(* PLC project Unbenannt, Unbekannt Unbenannt 1 *)
(* stored: creationDateTime 2019-08-23T13:38:07, modificationDateTime 2019-09-16T21:40:09 *)

(* Output current execution time in miliseconds *)
FUNCTION T_PLC_MS : UDINT
  VAR
    tx : UDINT;
  END_VAR
  VAR_INPUT
    debug : BOOL;
  END_VAR
  VAR
    N : INT := 0;
    offset : UDINT := 0;
    temp : DWORD := 1;
  END_VAR

            tx := 0;

{extern unsigned long __tick;
extern unsigned long long common_ticktime__;
unsigned long long ticktime_ms = (common_ticktime__)/1000000;
UDINT plc_time = (UDINT)(ticktime_ms * (unsigned long long)__tick);
TX = plc_time}

T_PLC_MS := tx;
IF debug THEN
	T_PLC_MS := (DWORD_TO_UDINT(SHL(UDINT_TO_DWORD(T_PLC_MS),N) OR SHL(temp,N))-1) + OFFSET;
END_IF;

(* Original Code:
tx := TIME();
T_PLC_MS := TIME_TO_DWORD(Tx);
IF debug THEN
	T_PLC_MS := (SHL(T_PLC_MS,N) OR SHL(DWORD#1,N)-1) + OFFSET;
END_IF;
*)

(* From OSCAT library, www.oscat.de

this is a temporary T_PLC_MS FB until OpenPLC gets it´s own time() functionality *)

(* PLC_TIME and Global variables PLC_SCAN_CYCL and PLC_CYCL_TIME required *)
          
END_FUNCTION

FUNCTION_BLOCK F_POLY
  VAR_INPUT
    X : REAL;
    C : ARRAY[0..7] OF REAL;
  END_VAR
  VAR_OUTPUT
    _F_POLY : REAL;
  END_VAR

            _F_POLY := ((((((( c[7] * x + c[6] ) * x + c[5] ) * x + c[4] ) * x + c[3] ) * x + c[2] ) * x + c[1] ) * x + c[0] ) ;

          
END_FUNCTION_BLOCK

PROGRAM program0
  VAR
    LocalVar0 : DINT;
    LocalVar1 : DINT;
    LocalVar2 : DINT;
    LocalVar3 : REAL;
    F_POLY0 : F_POLY;
  END_VAR

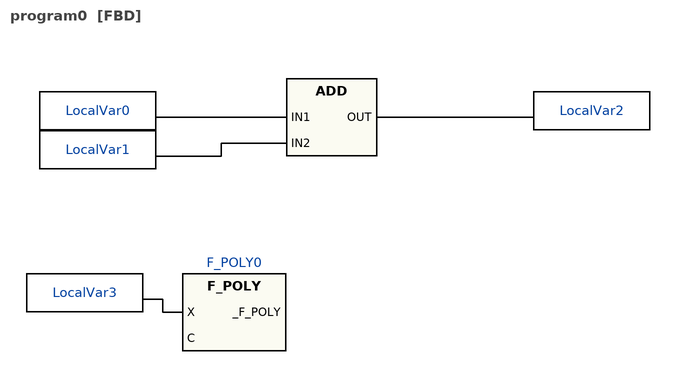
(* FBD diagram, written out as Structured Text *)
LocalVar2 := LocalVar0 + LocalVar1;
F_POLY0(X := LocalVar3);
END_PROGRAM

(* calculates the linear equation f_lin = a*x + b *)
FUNCTION F_LIN : REAL
  VAR_INPUT
    X : REAL;
    A : REAL;
    B : REAL;
  END_VAR

            F_lin := A * X + B;
(* from OSCAT library www.oscat.de *)
          
END_FUNCTION

(* this function calculates the linear equation f_lin = a*x + b given by two points x1/y1 and x2/y2 *)
FUNCTION F_LIN2 : REAL
  VAR_INPUT
    X : REAL;
    X1 : REAL;
    X2 : REAL;
    Y1 : REAL;
    Y2 : REAL;
  END_VAR

            F_LIN2 := (Y2 - Y1) / (X2 - X1) * (X - X1) + Y1;
(* from OSCAT library www.oscat.de *)
          
END_FUNCTION

(* calculates the power equation f_power = a*x^n *)
FUNCTION F_POWER : REAL
  VAR
    A : REAL;
    X : REAL;
    N : REAL;
  END_VAR

            f_power := a * EXPT(X,N);
(* from OSCAT library www.oscat.de *)
          
END_FUNCTION

(* calculates the quadratic equation f_lin = a*x + b *)
FUNCTION F_QUAD : REAL
  VAR
    X : REAL;
    A : REAL;
    B : REAL;
    C : REAL;
  END_VAR

            F_QUAD :=  (A * X + B) * X + C;
(* from OSCAT library www.oscat.de *)
          
END_FUNCTION

(* calculates a ramp and limits the output to 0 .. 255 without overflow problems *)
FUNCTION FRMP_B : BYTE
  VAR
    START : BYTE;
    DIR : BOOL;
    TD : TIME;
    TR : TIME;
  END_VAR

            IF TD < TR THEN
	FRMP_B := MIN(UDINT_TO_BYTE(DWORD_TO_UDINT(SHL(TIME_TO_DWORD(TD), 8)) / TIME_TO_UDINT(TR)), SEL(DIR, START, USINT_TO_BYTE(USINT#255 - BYTE_TO_USINT(START))));
	IF DIR THEN
		FRMP_B := USINT_TO_BYTE(BYTE_TO_USINT(START) + BYTE_TO_USINT(FRMP_B));
	ELSE
		FRMP_B := USINT_TO_BYTE(BYTE_TO_USINT(START) - BYTE_TO_USINT(FRMP_B));
	END_IF;
ELSE
	FRMP_B := SEL(DIR, BYTE#0, BYTE#255);
END_IF;
(* from OSCAT library www.oscat.de *)
          
END_FUNCTION

(* This is a increment function which increments the variable X by 1 and if N is reached, it begins with 0 instead of N again. *)
FUNCTION INC1 : INT
  VAR_INPUT
    X : INT;
    N : INT;
  END_VAR

            IF X >= N - 1 THEN
	INC1 := 0;
ELSE
	INC1 := X + 1;
END_IF;
(* from OSCAT library www.oscat.de *)
          
END_FUNCTION

(* this function block delays input values by each programm cycle after N+1 cycles the in value has shifted to the out. N can be any alue from 0 .. 32 if n = 0 the input will be present on the output without a delay. f N > 32 then the output will be delayed by 32 cycles. any high on rst will load the buffer with in. *)
FUNCTION_BLOCK DELAY
  VAR_INPUT
    IN : REAL;
    N : INT;
    RST : BOOL;
  END_VAR
  VAR_OUTPUT
    OUT : REAL;
  END_VAR
  VAR
    i : INT;
    init : BOOL;
    stop : INT;
    buf : ARRAY[0..31] OF REAL;
  END_VAR

            stop := LIMIT(0,N,32) - 1;
IF rst OR NOT init THEN
	init := TRUE;
	FOR i := 0 TO stop DO buf[i] := in; END_FOR;
	out := in;
	i := 0;
ELSIF stop < 0 THEN
	out := in;
ELSE
	out := buf[i];
	buf[i] := in;
	i := INC1(i, N);
END_IF;
(* from OSCAT library www.oscat.de *)
(* inc1 requiered *)
          
END_FUNCTION_BLOCK

(* this function calculates the moving average over n samples from a sequential input the input values are shifted into an N deep buffer and the avg of this buffer is diplayed at anytime on the output. a rst will load the buffer with the current in value.. *)
FUNCTION_BLOCK FT_AVG
  VAR_INPUT
    IN : REAL;
    _E : BOOL := TRUE;
    RST : BOOL;
    N : INT := 32;
  END_VAR
  VAR_OUTPUT
    AVG : REAL;
  END_VAR
  VAR
    buff : DELAY;
    i : INT;
    init : BOOL;
  END_VAR

            buff.N := LIMIT(0, N, 32);

IF NOT init OR rst THEN
	FOR i := 1 TO N DO
		buff(in := in);
	END_FOR;
	avg := in;
	init := TRUE;
ELSIF _E THEN
	buff(in := in);
	avg := avg + (in - buff.out ) / INT_TO_REAL(N);
END_IF;
(* from OSCAT library www.oscat.de *)
(* FB FC delay and inc1 requiered *)
          
END_FUNCTION_BLOCK

(* this function block stores the min and max value of an input signal. when rst is true the mn and mx outputs are set to the in value. when a rst is never active the function autoresets to the in value at startup. since the input might not be present at first cycle the mn and mx are set during second cycle. *)
FUNCTION_BLOCK FT_MIN_MAX
  VAR_INPUT
    IN : REAL;
    RST : BOOL;
  END_VAR
  VAR_OUTPUT
    MX : REAL;
    MN : REAL;
  END_VAR
  VAR
    init : BOOL;
  END_VAR

            IF (rst = TRUE) OR (init = FALSE) THEN
  mn := in;
  mx := in;
  init := TRUE;
ELSIF (in < mn) THEN
  mn := in;
ELSIF (in > mx) THEN
  mx := in;
END_IF;
(* from OSCAT library www.oscat.de *)
          
END_FUNCTION_BLOCK

(* LINEAR_INT calculates an output based on a linear interpolation of up to 20 coordinates given in an array the input coordinates have to start at the lowest array position and must be sorted ba ascending X values. *)
FUNCTION LINEAR_INT : REAL
  VAR_INPUT
    X : REAL;
    XY : ARRAY[1..20, 0..1] OF REAL;
    Pts : INT;
  END_VAR
  VAR
    i : INT;
  END_VAR

            pts := MIN(pts,20);
i := 2;
WHILE (i < pts) AND (XY[i,0] < X) DO
	i := i + 1;
END_WHILE;
LINEAR_INT := ((XY[i,1] - XY[i-1,1]) * X - XY[i,1] * XY[i-1,0] + XY[i-1,1] * XY[i,0]) / (XY[i,0] - XY[i-1,0]);
(* from OSCAT library www.oscat.de *)
          
END_FUNCTION

(* POLYNOM_INT calculates an output based on a Polynom interpolation of up to 5 coordinates given in an array the indut coordinates have to start at the lowest array position and must be sorted ba ascending X values. *)
FUNCTION POLYNOM_INT : REAL
  VAR_INPUT
    X : REAL;
    XY : ARRAY[1..5, 0..1] OF REAL;
    Pts : INT;
  END_VAR
  VAR
    I : INT;
    J : INT;
    stop : INT;
  END_VAR

            pts := MIN(pts, 5);
FOR i := 1 TO pts DO
	stop := i + 1;
   	FOR j := pts TO stop BY -1 DO
   		XY[j,1] := (XY[j,1] - XY[j-1,1]) / (XY[j,0] - XY[j-i,0]);
	END_FOR;
END_FOR;
POLYNOM_INT := 0.0;
FOR i := pts TO 1 BY -1 DO
       POLYNOM_INT := POLYNOM_INT * (X - XY[i,0]) + XY[i,1];
END_FOR;


          
END_FUNCTION

(* this ramp function follows an input signal with a linear ramp up or down, the up or down speed can be set with KF and KR. a K factor of 1 means 1 unit per second on the output. K factors can only be positive and not negative. a busy output signals the ramp is running or busy false means the in value is present on the output. a rmp input false means the output follows the input dierctly while a rmp = true means the output follows the input with a ramp. a updn output signal the directon of the ramp (up or down). *)
FUNCTION_BLOCK FT_RMP
  VAR_INPUT
    RMP : BOOL := TRUE;
    IN : REAL;
    KR : REAL;
    KF : REAL;
  END_VAR
  VAR_OUTPUT
    OUT : REAL;
    BUSY : BOOL;
    UD : BOOL;
  END_VAR
  VAR
    tx : TIME;
    last : TIME;
    init : BOOL;
  END_VAR

            
tx := UDINT_TO_TIME(T_PLC_MS(en:=true)) - last;

IF NOT init THEN
	init := TRUE;
	last := tx;
	tx := t#0s;
	out := in;
END_IF;
IF NOT rmp THEN
	out := in;
	busy := FALSE;
ELSIF out > in THEN
	(* ramp down *)
	out := out - TIME_TO_REAL(tx) * 0.001 * KF;
	out := MAX(in, out);
ELSIF out < in THEN
	(* ramp up *)
	out := out + TIME_TO_REAL(tx) * 0.001 * KR;
	out := MIN(in, out);
END_IF;

(* set busy and dir flags *)
IF out < in THEN
	busy := TRUE;
	ud := TRUE;
ELSIF out > in THEN
	busy := TRUE;
	ud := FALSE;
ELSE
	busy := FALSE;
END_IF;
last := last + tx;

(* From Oscat Library, www.oscat.de *)
          
END_FUNCTION_BLOCK

FUNCTION_BLOCK _FB_LINEAR_INT
  VAR_INPUT
    X : REAL;
    XY : ARRAY[1..20, 0..1] OF REAL;
    PTS : INT;
  END_VAR
  VAR_OUTPUT
    _LINEAR_INT : REAL;
  END_VAR
  VAR
    i : INT;
    i2 : INT;
  END_VAR

            pts := MIN(pts,20);

i := 2;

WHILE (i < pts) AND (XY[i,0] < X) DO

	i := i + 1;

END_WHILE;

_LINEAR_INT := ((XY[i,1] - XY[i-1,1]) * X - XY[i,1] * XY[i-1,0] + XY[i-1,1] * XY[i,0]) / (XY[i,0] - XY[i-1,0]);




(* From OSCAT Library, www.oscat.de *)
          
END_FUNCTION_BLOCK

CONFIGURATION Config0
  RESOURCE Res0 ON PLC
    TASK task0(INTERVAL := T#20ms, PRIORITY := 0);
    PROGRAM instance0 WITH task0 : program0;
  END_RESOURCE
END_CONFIGURATION
